TYPE st_RobotWarehouseMove_Status :
STRUCT
	bBusy	: BOOL;
	bDone	: BOOL;
	bError	: BOOL;
	iErrorID : UDINT;
	Status : STRING;
END_STRUCT
END_TYPE

(* stored: Version 1.1.0.1, ProductVersion 3.1.4024.13
   DUT st_RobotWarehouseMove_Status: Id {9e40a5cc-b3b7-4653-bbb3-426b8c3b4a40} *)
